(* IEC 61131-3 sources: jiepp/tests/jiepp/input/line_macro, 6 files *)

(* ---- a.iec ---- *)
program a0
__LINE__;
end_program

{#include "b.iec"}

program a1
__LINE__;
end_program

(* ---- b.iec ---- *)
__LINE__;{#include "c.iec"};__LINE__;

program b
__LINE__;
end_program

(* ---- c.iec ---- *)
program c
__LINE__;
end_program

(* ---- line_macro_fmacro.iec ---- *)
{#define F(x, y) $
    x $
    + $
    y $
}
{#define  $
    G(    $
        x $
        , $
        y $
    )     $
          $
    F(    $
    x * y $
    ,     $
    x / y $
    )     $
}

program Main

__LINE__;
(F(
    2,
    3)) ** (G(
    4,
    5));
__LINE__;

end_program

(* ---- line_macro_include.iec ---- *)
{#include "a.iec"}

program X
__LINE__;
end_program

(* ---- line_macro_omacro.iec ---- *)
{#define M $
    2$
    $
}

{#define $
    N $
    $
    3$
    $
    $
}

program Main

__LINE__;
M
+
N;
__LINE__;

end_program
